// TwinCAT 3 PLC project UnitTest
// Title: TestFramework
// Company: Hoox.Software
// Author: Patrick Dressel
// ProjectVersion: 2.1.0
// ProgramVersion: 3.1.4022.6
// libraries:
//   Tc2_Standard, * (Beckhoff Automation GmbH)
//   Tc2_System, * (Beckhoff Automation GmbH)
//   Tc2_Utilities, * (Beckhoff Automation GmbH)
//   Tc3_Module, * (Beckhoff Automation GmbH)
//   Base Interfaces,newest,System
// project tree:
//   Datatypes/ EResult_t.TcDUT (not stored), EAssertion_t.TcDUT, ERetCode_t.TcDUT (not stored), EState_t.TcDUT (not stored), IdHandle_t.TcDUT (not stored), ObjectId_t.TcDUT (not stored), SStatistic_t.TcDUT (not stored), STestcase_t.TcDUT (not stored), StringHandle_t.TcDUT, StrMessage_t.TcDUT, TestCaseHandle_t.TcDUT (not stored)
//   Datatypes/Report/ EExportState_t.TcDUT (not stored), EReportType_t.TcDUT (not stored), NameHandle_t.TcDUT (not stored), PathHandle_t.TcDUT (not stored), StrFileName_t.TcDUT, StrPathName_t.TcDUT (not stored), TestReportHandle_t.TcDUT (not stored), UBaseTypes_t.TcDUT, UTime_t.TcDUT
//   GVLs/ GVL_Parameter.TcGVL (not stored), GVL_Sample.TcGVL (not stored) (excluded from build)
//   / PlcTask.TcTTO
//   Source/ FB_Assertion.TcPOU (not stored), FB_Testsuite.TcPOU (not stored), FB_TestBase.TcPOU, ITestBase_t.TcIO, ITestsuite_t.TcIO (not stored), PRG_TestLib.TcPOU
//   Source/Report/ FB_CoverageFile.TcPOU (not stored), FB_TestReportBase.TcPOU, FB_FileBase.TcPOU (not stored), FB_TextReport.TcPOU (not stored)
//   Test/ FB_Test_Base.TcPOU, FB_Test_Base_Ptr.TcPOU (not stored), FB_Test_Base_Not.TcPOU (not stored), FB_Test_Base_Delay.TcPOU

CONFIGURATION UnitTest
    RESOURCE PLC ON TwinCAT3
        TASK PlcTask(INTERVAL := T#10ms, PRIORITY := 20);
    END_RESOURCE
END_CONFIGURATION

// ---- Datatypes/EAssertion_t.TcDUT
{attribute 'qualified_only'}
{attribute 'strict'}
TYPE EAssertion_t :
(
	eStatePassed,
	eStateFailed,
	eStateFailedFatal
);
END_TYPE

// ---- Datatypes/Report/StrFileName_t.TcDUT
TYPE StrFileName_t : String(255); END_TYPE

// ---- Datatypes/Report/UBaseTypes_t.TcDUT
TYPE UBaseTypes_t :
UNION
	u8Value 	: USINT;
	s8Value 	: SINT;
	u16Value 	: UINT;
	s16Value 	: INT;
	u32Value 	: UDINT;
	s32Value 	: DINT;
	w16Value    : WORD;
	w32Value    : DWORD;
	r32Value 	: REAL;
	bValue		: BOOL;
END_UNION
END_TYPE

// ---- Datatypes/Report/UTime_t.TcDUT
TYPE UTime_t :
UNION
	dwValue  : ARRAY[0..1] OF DWORD;
	u64Value : ULINT;
END_UNION
END_TYPE

// ---- Datatypes/StringHandle_t.TcDUT
TYPE StringHandle_t : POINTER TO String(255); END_TYPE

// ---- Datatypes/StrMessage_t.TcDUT
TYPE StrMessage_t : String(255); END_TYPE

// ---- Source/ITestBase_t.TcIO
INTERFACE ITestBase_t

METHOD PUBLIC _cleanup : ERetCode_t
VAR_INPUT
END_VAR
END_METHOD

METHOD PUBLIC _execute : ERetCode_t
VAR_INPUT
END_VAR
END_METHOD

METHOD PUBLIC _prepare : ERetCode_t
VAR_INPUT
END_VAR
END_METHOD

METHOD getClassname : ObjectId_t
VAR_INPUT
END_VAR
END_METHOD

METHOD getId : ObjectId_t
VAR_INPUT
END_VAR
END_METHOD

METHOD getMessage : StrMessage_t
VAR_INPUT
END_VAR
END_METHOD

METHOD getPath : ObjectId_t
VAR_INPUT
END_VAR
END_METHOD

PROPERTY Result : STestcase_t
GET
END_GET
END_PROPERTY

END_INTERFACE

// ---- Source/FB_TestBase.TcPOU
(******************************************************************************
Baustein: FB_TestBase
Spezifikation: doc/Spezifikation.pdf, Kap. x.y.z
-------------------------------------------------------------------------------
erstellt:
von:
Geändert:
von:
-------------------------------------------------------------------------------
Beschreibung
Dieser Baustein stellt die Basis für einen Unittest dar und enthält
alle notwendigen Variablen und Methoden zur Testauswertung.

-------------------------------------------------------------------------------
Input
-

Output
	o_eResult: EResult_t;
******************************************************************************)
FUNCTION_BLOCK FB_TestBase
    IMPLEMENTS ITestBase_t
VAR_INPUT
END_VAR
VAR_OUTPUT
	o_eResult       : EResult_t;
END_VAR
VAR
	strId	  		: ObjectId_t;
	strClassName	: ObjectId_t;
	strPath			: ObjectId_t;
	strMessage 	 	: StrMessage_t;
	u32StartTime	: UDINT;
	u32EndTime		: UDINT;
	iTestSuite      : ITestsuite_t;
	bRegistered 	: BOOL;
    sResult         : STestcase_t;
    assert          : FB_Assertion;
END_VAR

(******************************************************************************
Baustein: FB_TestBase.cleanup
Spezifikation: doc/Spezifikation.pdf, Kap. x.y.z
-------------------------------------------------------------------------------
erstellt:
von:
Geändert:
von:
-------------------------------------------------------------------------------
Beschreibung
Diese Methode...

-------------------------------------------------------------------------------
Input
-

Output
-
******************************************************************************)
{attribute 'hide'} 
METHOD PUBLIC FINAL _cleanup : ERetCode_t
VAR_INPUT
END_VAR


	_cleanup := cleanup();

    IF _cleanup = ERetCode_t.eRetDone THEN
        setEndTime();
    END_IF;	
	
    CASE assert.o_eState OF 

    EAssertion_t.eStateFailed:
        o_eResult := EResult_t.eStateFailed;

    EAssertion_t.eStateFailedFatal:
        o_eResult := EResult_t.eStateFailedFatal;

    END_CASE;
END_METHOD

(******************************************************************************
Baustein: FB_TestBase.execute
Spezifikation: doc/Spezifikation.pdf, Kap. x.y.z
-------------------------------------------------------------------------------
erstellt:
von:
Geändert:
von:
-------------------------------------------------------------------------------
Beschreibung
Diese Methode...

-------------------------------------------------------------------------------
Input
-

Output
-
******************************************************************************)
{attribute 'hide'} 
METHOD PUBLIC FINAL _execute : ERetCode_t
VAR_INPUT
END_VAR

	_execute := execute();
END_METHOD

(******************************************************************************
Baustein: FB_TestBase.prepare
Spezifikation: doc/Spezifikation.pdf, Kap. x.y.z
-------------------------------------------------------------------------------
erstellt:
von:
Geändert:
von:
-------------------------------------------------------------------------------
Beschreibung
Diese Methode...

-------------------------------------------------------------------------------
Input
-

Output
-
******************************************************************************)
{attribute 'hide'} 
METHOD PUBLIC FINAL _prepare : ERetCode_t
VAR_INPUT
END_VAR

	sResult.u32Passed 		:= 0;
	sResult.u32Failed 		:= 0;
	u32StartTime 	        := 0;
	u32EndTime 		        := 0;
	o_eResult 		        := EResult_t.eStateIdle;

	_prepare := prepare();

    IF _prepare = ERetCode_t.eRetDone THEN
        setStartTime();
    END_IF;
END_METHOD

(******************************************************************************
Baustein: FB_TestBase.cleanup
Spezifikation: doc/Spezifikation.pdf, Kap. x.y.z
-------------------------------------------------------------------------------
erstellt:
von:
Geändert:
von:
-------------------------------------------------------------------------------
Beschreibung
Diese Methode...

-------------------------------------------------------------------------------
Input
-

Output
-
******************************************************************************)
METHOD PUBLIC cleanup : ERetCode_t
VAR_INPUT
END_VAR

	cleanup := ERetCode_t.eRetFailed;
END_METHOD

(******************************************************************************
Baustein: FB_TestBase.execute
Spezifikation: doc/Spezifikation.pdf, Kap. x.y.z
-------------------------------------------------------------------------------
erstellt:
von:
Geändert:
von:
-------------------------------------------------------------------------------
Beschreibung
Diese Methode...

-------------------------------------------------------------------------------
Input
-

Output
-
******************************************************************************)
METHOD PUBLIC execute : ERetCode_t
VAR_INPUT
END_VAR

	Execute := ERetCode_t.eRetFailed;
END_METHOD

(******************************************************************************
Baustein: FB_Testsuite.FB_init
Spezifikation: doc/Spezifikation.pdf, Kap. x.y.z
-------------------------------------------------------------------------------
erstellt:
von:
Geändert:
von:
-------------------------------------------------------------------------------
Beschreibung
Diese Methode

-------------------------------------------------------------------------------
Input
-

Output
-
******************************************************************************)
{attribute 'hide'} 
METHOD FB_init : BOOL
VAR_INPUT
	bInitRetains 	: BOOL; // if TRUE, the retain variables are initialized (warm start / cold start)
	bInCopyCode 	: BOOL;  // if TRUE, the instance afterwards gets moved into the copy code (online change)
	i_strId	  		: ObjectId_t;
	i_strClassName	: ObjectId_t;
	i_strPath 		: ObjectId_t;
	i_iTestSuite 	: ITestSuite_t;
	i_bExecute      : BOOL := true; 
END_VAR
	
	strId 		 := i_strId;
	strClassName := i_strClassName;
	strPath 	 := i_strPath;
	iTestSuite 	 := i_iTestSuite;

    IF i_bExecute = FALSE THEN
        o_eResult := EResult_t.eStateSkipped;
    END_IF;
	
	register();
END_METHOD

(******************************************************************************
Baustein: FB_TestBase.getId
Spezifikation: doc/Spezifikation.pdf, Kap. x.y.z
-------------------------------------------------------------------------------
erstellt:
von:
Geändert:
von:
-------------------------------------------------------------------------------
Beschreibung
Diese Methode

-------------------------------------------------------------------------------
Input
-

Output
-
******************************************************************************)
{attribute 'hide'} 
METHOD PUBLIC FINAL getClassName : ObjectId_t
VAR_INPUT
END_VAR

	getClassName := strClassName;
END_METHOD

(******************************************************************************
Baustein: FB_TestBase.getFailed
Spezifikation: doc/Spezifikation.pdf, Kap. x.y.z
-------------------------------------------------------------------------------
erstellt:
von:
Geändert:
von:
-------------------------------------------------------------------------------
Beschreibung
Diese Methode

-------------------------------------------------------------------------------
Input
-

Output
-
******************************************************************************)
{attribute 'hide'} 
METHOD PUBLIC FINAL getFailed : UDINT
VAR_INPUT
END_VAR

	getFailed := assert.o_u32Failed;
END_METHOD

(******************************************************************************
Baustein: FB_TestBase.getId
Spezifikation: doc/Spezifikation.pdf, Kap. x.y.z
-------------------------------------------------------------------------------
erstellt:
von:
Geändert:
von:
-------------------------------------------------------------------------------
Beschreibung
Diese Methode

-------------------------------------------------------------------------------
Input
-

Output
-
******************************************************************************)
{attribute 'hide'} 
METHOD PUBLIC FINAL getId : ObjectId_t
VAR_INPUT
END_VAR

	getId := strId;
END_METHOD

METHOD PUBLIC FINAL getMessage : StrMessage_t
VAR_INPUT
END_VAR

	getMessage := strMessage;
END_METHOD

(******************************************************************************
Baustein: FB_TestBase.getPassed
Spezifikation: doc/Spezifikation.pdf, Kap. x.y.z
-------------------------------------------------------------------------------
erstellt:
von:
Geändert:
von:
-------------------------------------------------------------------------------
Beschreibung
Diese Methode

-------------------------------------------------------------------------------
Input
-

Output
-
******************************************************************************)
{attribute 'hide'} 
METHOD PUBLIC FINAL getPassed : UDINT
VAR_INPUT
END_VAR

	getPassed := assert.o_u32Passed;
END_METHOD

(******************************************************************************
Baustein: FB_TestBase.getPassed
Spezifikation: doc/Spezifikation.pdf, Kap. x.y.z
-------------------------------------------------------------------------------
erstellt:
von:
Geändert:
von:
-------------------------------------------------------------------------------
Beschreibung
Diese Methode

-------------------------------------------------------------------------------
Input
-

Output
-
******************************************************************************)
{attribute 'hide'} 
METHOD PUBLIC FINAL getPath : ObjectId_t
VAR_INPUT
END_VAR

	getPath := strPath;
END_METHOD

(******************************************************************************
Baustein: FB_TestBase.getPassed
Spezifikation: doc/Spezifikation.pdf, Kap. x.y.z
-------------------------------------------------------------------------------
erstellt:
von:
Geändert:
von:
-------------------------------------------------------------------------------
Beschreibung
Diese Methode

-------------------------------------------------------------------------------
Input
-

Output
-
******************************************************************************)
{attribute 'hide'} 
METHOD PRIVATE FINAL getSystemTime : UDINT
VAR_INPUT
END_VAR
VAR
	u64Time : ULINT;
END_VAR

	u64Time := F_GetSystemTime()/10000;


	getSystemTime := to_udint(u64Time and 16#FFFFFFFF);
END_METHOD

(******************************************************************************
Baustein: FB_TestBase.getPassed
Spezifikation: doc/Spezifikation.pdf, Kap. x.y.z
-------------------------------------------------------------------------------
erstellt:
von:
Geändert:
von:
-------------------------------------------------------------------------------
Beschreibung
Diese Methode

-------------------------------------------------------------------------------
Input
-

Output
-
******************************************************************************)
{attribute 'hide'} 
METHOD PUBLIC FINAL getTime : UDINT
VAR_INPUT
END_VAR

	getTime := 0;

	IF u32EndTime > u32StartTime THEN
		getTime := u32EndTime - u32StartTime;
	END_IF;
END_METHOD

(******************************************************************************
Baustein: FB_TestBase.logError
Spezifikation: doc/Spezifikation.pdf, Kap. x.y.z
-------------------------------------------------------------------------------
erstellt:
von:
Geändert:
von:
-------------------------------------------------------------------------------
Beschreibung
Diese Methode

-------------------------------------------------------------------------------
Input
-

Output
-
******************************************************************************)
{attribute 'hide'} 
METHOD PROTECTED FINAL logError : BOOL
VAR_INPUT
	i_strMessage : StrMessage_t;
END_VAR

	ADSLOGSTR(msgCtrlMask 	:= ADSLOG_MSGTYPE_ERROR , 
			  msgFmtStr 	:= i_strMessage, 
			  strArg 		:= '');
END_METHOD

(******************************************************************************
Baustein: FB_TestBase.logInfo
Spezifikation: doc/Spezifikation.pdf, Kap. x.y.z
-------------------------------------------------------------------------------
erstellt:
von:
Geändert:
von:
-------------------------------------------------------------------------------
Beschreibung
Diese Methode

-------------------------------------------------------------------------------
Input
-

Output
-
******************************************************************************)
{attribute 'hide'} 
METHOD INTERNAL FINAL logInfo : BOOL
VAR_INPUT
	i_strMessage : StrMessage_t;
END_VAR

	ADSLOGSTR(msgCtrlMask 	:= ADSLOG_MSGTYPE_HINT , 
			  msgFmtStr 	:= i_strMessage, 
			  strArg 		:= '');
END_METHOD

(******************************************************************************
Baustein: FB_TestBase.prepare
Spezifikation: doc/Spezifikation.pdf, Kap. x.y.z
-------------------------------------------------------------------------------
erstellt:
von:
Geändert:
von:
-------------------------------------------------------------------------------
Beschreibung
Diese Methode...

-------------------------------------------------------------------------------
Input
-

Output
-
******************************************************************************)
METHOD PUBLIC prepare : ERetCode_t
VAR_INPUT
END_VAR

	prepare := ERetCode_t.eRetFailed;
END_METHOD

(******************************************************************************
Baustein: FB_TestBase.register
Spezifikation: doc/Spezifikation.pdf, Kap. x.y.z
-------------------------------------------------------------------------------
erstellt:
von:
Geändert:
von:
-------------------------------------------------------------------------------
Beschreibung
Diese Methode

-------------------------------------------------------------------------------
Input
-

Output
-
******************************************************************************)
{attribute 'hide'} 
METHOD INTERNAL FINAL register : BOOL
VAR_INPUT
END_VAR

	IF iTestSuite <> 0 	AND 
       bRegistered = FALSE  THEN
		
	   bRegistered := iTestSuite.addTestcase(THIS^);
	
	END_IF
END_METHOD

{warning 'Eigenschaftenimplementierung hinzufügen'}
PROPERTY Result : STestcase_t
GET

    sResult.u32Time := getTime();
    sResult.eState  := o_eResult; 
    Result          := sResult;
END_GET
END_PROPERTY

(******************************************************************************
Baustein: FB_TestBase.getPassed
Spezifikation: doc/Spezifikation.pdf, Kap. x.y.z
-------------------------------------------------------------------------------
erstellt:
von:
Geändert:
von:
-------------------------------------------------------------------------------
Beschreibung
Diese Methode

-------------------------------------------------------------------------------
Input
-

Output
-
******************************************************************************)
{attribute 'hide'} 
METHOD INTERNAL FINAL setEndTime : BOOL
VAR_INPUT
END_VAR

	IF u32EndTime = 0 THEN
		u32EndTime := getSystemTime();
	END_IF;
	setEndTime := true;
END_METHOD

METHOD PROTECTED FINAL setMessage
VAR_INPUT
	strValue : StrMessage_t;
END_VAR

	IF o_eResult < EResult_t.eStateFailed THEN
		strMessage := strValue;
	END_IF;
END_METHOD

(******************************************************************************
Baustein: FB_TestBase.getPassed
Spezifikation: doc/Spezifikation.pdf, Kap. x.y.z
-------------------------------------------------------------------------------
erstellt:
von:
Geändert:
von:
-------------------------------------------------------------------------------
Beschreibung
Diese Methode

-------------------------------------------------------------------------------
Input
-

Output
-
******************************************************************************)
{attribute 'hide'} 
METHOD INTERNAL FINAL setStartTime : BOOL
VAR_INPUT
END_VAR

	IF u32StartTime = 0 THEN
		u32StartTime   	:= getSystemTime();
	END_IF;
	setStartTime := true;
END_METHOD

(******************************************************************************
Baustein: FB_TestBase.strncmp
Spezifikation: doc/Spezifikation.pdf, Kap. x.y.z
-------------------------------------------------------------------------------
erstellt:
von:
Geändert:
von:
-------------------------------------------------------------------------------
Beschreibung
Diese Methode

-------------------------------------------------------------------------------
Input
	strInput 	: StringHandle_t;
	strCompare 	: StringHandle_t;
	s16Size		: INT;

Output
-
******************************************************************************)
{attribute 'hide'} 
METHOD PRIVATE FINAL strncmp : BOOL
VAR_INPUT
	strInput 	: StringHandle_t;
	strCompare 	: StringHandle_t;
	s16Size		: INT;
END_VAR
VAR
	s16Size1 : INT;
	s16Size2 : INT;
	s16Diff  : INT;
END_VAR

   s16Size1:= LEN(strInput^); 
	s16Size2:= LEN(strCompare^); 
	
	strncmp := FALSE;
	
	s16Diff := s16Size1 - s16Size2;
   
	// vergleich nur wenn beide Strings
	// gleich groß sind.
	IF s16Diff  = 0 THEN

		strncmp := TRUE;
	
		WHILE(s16Size > 0) DO

			IF strInput^ <> strCompare^ THEN
				strncmp := FALSE;
			END_IF;  
 
			strInput   := strInput + 1;
			strCompare := strCompare + 1;
			s16Size    := s16Size - 1;

		END_WHILE


	
	END_IF;
END_METHOD

(******************************************************************************
Baustein: FB_TestBase.validate
Spezifikation: doc/Spezifikation.pdf, Kap. x.y.z
-------------------------------------------------------------------------------
erstellt:
von:
Geändert:
von:
-------------------------------------------------------------------------------
Beschreibung
Diese Methode

-------------------------------------------------------------------------------
Input
	var1 : ANY;
	var2 : ANY;

Output
-
******************************************************************************)
{attribute 'hide'} 
METHOD PRIVATE FINAL validate : BOOL
VAR_INPUT
	var1 : ANY;
	var2 : ANY;
END_VAR

	validate := FALSE;
	
	IF (var1.pValue = 0 OR var2.pValue = 0) THEN
		logError(concat('Assert validation fails with NULL-Pointer: ', strId));
		RETURN;
	END_IF

	IF (var1.TypeClass <> var2.TypeClass) THEN
		logError(concat('Assert validation fails with TypeClass Error: ', strId));
		RETURN;
	END_IF;	
	
	IF (var1.diSize <> var2.diSize) THEN
		logError(concat('Assert validation fails with different size: ', strId));
		RETURN;
	END_IF;	
	
	validate := true;
END_METHOD

END_FUNCTION_BLOCK

// ---- Source/PRG_TestLib.TcPOU
(******************************************************************************
Baustein: PRG_TestLibrary
Spezifikation: doc/Spezifikation.pdf, Kap. x.y.z
-------------------------------------------------------------------------------
erstellt:
von:
Geändert:
von:
-------------------------------------------------------------------------------
Beschreibung
Dieser Baustein etnhält alle Testsuites und führt diese aus.

-------------------------------------------------------------------------------
Input
	i_bStart : mit positiver Flanke werden die registrierten Testsuites ausgeführt

Output
	o_eState  		: EState_t;
	o_eResult 		: EResult_t;
	o_sStatistic	: SStatistic_t;
******************************************************************************)
{attribute 'global_init_slot' := '41000'}
PROGRAM PRG_TestLib
VAR_INPUT
	i_bStart : BOOL;
END_VAR
VAR_OUTPUT
	o_eState  		: EState_t;
	o_eResult 		: EResult_t;
	o_sStatistic	: SStatistic_t;
END_VAR
VAR
	bHwStart AT %I* : BOOL;
	bHwBusy  AT %Q* : BOOL;
	bHwReady AT %Q* : BOOL;
	
	a_iTestSuite 	: ARRAY [0..255] OF ITestSuite_t;
	u16TestSuites 	: UINT;
	u16Index	  	: UINT;
	iActTestSuite 	: ITestSuite_t;
	pTestReport		: POINTER TO FB_TestReportBase;
	eRetCode 		: ERetCode_t;

	fbSystemTime 	: FB_LocalSystemTime;
	
	fbUnittest 		: FB_CoverageFile;
	u16ReportState  : UINT;
	u16TestSuitIdx	: UINT;
	iTestCase  		: ITestBase_t;
	sTempResult     : SStatistic_t;
END_VAR
VAR CONSTANT 
END_VAR


	fbSystemTime(bEnable := TRUE, dwCycle := 5);
			
	fbUnittest();

	CASE o_eState OF 
	
	EState_t.eStateInit:	
		
		IF i_bStart = FALSE THEN 
		   logInfo('Testlib V2.1.0 Ready');
			o_eState := EState_t.eStateIdle; 
		END_IF

	EState_t.eStateIdle:
	
		IF i_bStart = TRUE OR bHwStart = TRUE THEN
			logInfo('+++++++++++++ Testbeginn ++++++++++++++');
			o_eState := EState_t.eStatePrepare;
			bHwReady := FALSE;
		END_IF
	
	EState_t.eStatePrepare:
	
		bHwBusy := TRUE;
		
		o_eResult 	  				:= EResult_t.eStatePassed;
		o_sStatistic.u32Executed 	:= 0;
		o_sStatistic.u32TestCases	:= 0;
		o_sStatistic.u32Asserts  	:= 0;
		o_sStatistic.u32Passed   	:= 0;
		o_sStatistic.u32Failed	 	:= 0;	

		iActTestSuite := getFirstTestSuite();
		
		IF iActTestSuite      <> 0   THEN
			o_eState := EState_t.eStateExecute;
		ELSE
			o_eState := EState_t.eStateError;	
		END_IF
	
	EState_t.eStateExecute:
	
		iActTestSuite.execute(i_bStart := TRUE);
	
		IF iActTestSuite.getState() = EState_t.eStateReady THEN
			
			IF iActTestSuite.getResult() = EResult_t.eStateFailed THEN
				o_eResult := EResult_t.eStateFailed;
			END_IF
			
			iActTestSuite.execute(i_bStart := FALSE);
			sTempResult := iActTestSuite.Result;

			o_eState := EState_t.eStateCleanUp;

			o_sStatistic.u32Executed 	:= o_sStatistic.u32Executed  + sTempResult.u32Executed;
			o_sStatistic.u32TestCases	:= o_sStatistic.u32TestCases + sTempResult.u32TestCases; 
			o_sStatistic.u32Asserts  	:= o_sStatistic.u32Asserts   + sTempResult.u32Asserts;
			o_sStatistic.u32Passed   	:= o_sStatistic.u32Passed    + sTempResult.u32Passed;
			o_sStatistic.u32Failed	 	:= o_sStatistic.u32Failed    + sTempResult.u32Failed;
		END_IF
	
	EState_t.eStateCleanUp:
	
		IF iActTestSuite.getResult() = EResult_t.eStateFailedFatal THEN
			o_eResult := EResult_t.eStateFailedFatal;
			o_eState  := EState_t.eStateExport;
			logInfo('+++++++++++++ Fatal Error : Test Ende ++++++++++++++');
		ELSE
			
			iActTestSuite := getNextTestSuite();
						
			IF iActTestSuite <> 0 THEN
				o_eState := EState_t.eStateExecute;
			ELSE
				o_eState := EState_t.eStateExport;
				logInfo('+++++++++++++ Test Ende ++++++++++++++');
			END_IF		
			
		END_IF

	EState_t.eStateExport:

		IF createReport(EReporttype_t.eExternalReport) = ERetCode_t.eRetDone THEN
			o_eState := EState_t.eStateBuildUnitTestFile;
		END_IF;
		
	EState_t.eStateBuildUnitTestFile:

		IF createReport(EReporttype_t.eUnitTestReport) = ERetCode_t.eRetDone THEN
			o_eState := EState_t.eStateReady;
		END_IF;
		
	EState_t.eStateReady:

		bHwReady := TRUE;
		bHwBusy  := FALSE;
		IF i_bStart  = FALSE AND 
			bHwStart = FALSE THEN
			o_eState := EState_t.eStateIdle;
		END_IF		
		
	EState_t.eStateError,
	EState_t.eStateLicenseError:
	
		bHwBusy  := FALSE;
		o_eState := EState_t.eStateError;

	END_CASE

(******************************************************************************
Baustein: PRG_UnitTestLib.addTestReport
Spezifikation: doc/Spezifikation.pdf, Kap. x.y.z
-------------------------------------------------------------------------------
erstellt:
von:
Geändert:
von:
-------------------------------------------------------------------------------
Beschreibung
Diese Methode

-------------------------------------------------------------------------------
Input
i_pTestReport

Output
-
******************************************************************************)
{attribute 'hide'} 
METHOD PUBLIC addTestReport : BOOL
VAR_INPUT
	i_pTestReport : TestReportHandle_t;
END_VAR

	pTestReport := i_pTestReport;
END_METHOD

(******************************************************************************
Baustein: PRG_UnitTestLib.addTestSuite
Spezifikation: doc/Spezifikation.pdf, Kap. x.y.z
-------------------------------------------------------------------------------
erstellt:
von:
Geändert:
von:
-------------------------------------------------------------------------------
Beschreibung
Diese Methode

-------------------------------------------------------------------------------
Input
i_pTestSuite

Output
-
******************************************************************************)
{attribute 'hide'} 
METHOD PUBLIC addTestSuite : BOOL
VAR_INPUT
	i_iTestSuite : ITestSuite_t;
END_VAR
VAR
    sStatistic : SStatistic_t;
END_VAR

	addTestSuite := FALSE;

	IF 	i_iTestSuite  <> 0   AND 
		u16TestSuites <  255 THEN
		
		a_iTestSuite[u16TestSuites] := i_iTestSuite;
		sStatistic      := i_iTestSuite.Result;
		u16TestSuites   := u16TestSuites +1;
	
		o_sStatistic.u32TestSuites := o_sStatistic.u32TestSuites + 1;
		o_sStatistic.u32TestCases  := o_sStatistic.u32TestCases + sStatistic.u32TestCases;
		
		addTestSuite := TRUE;
	END_IF
END_METHOD

{attribute 'hide'} 
METHOD PRIVATE createReport : ERetCode_t
VAR_INPUT
	i_eReporttype : EReportType_t;
END_VAR
VAR
	eRetcode    : ERetCode_t;
	u32Temp     : UDINT;
    sTestResult : STestcase_t;
    sStatistic  : SStatistic_t;
END_VAR

	createReport := ERetCode_t.eRetBusy;

	CASE u16ReportState OF

	0: 
		IF i_eReporttype = EReportType_t.eUnitTestReport THEN
			u16ReportState := 20;
		END_IF;

		IF i_eReporttype = EReportType_t.eExternalReport THEN
			u16ReportState := 100;
		END_IF;

// +++++++++++++++++++++++++++++++++++++++++++++++++++++++++++
//
// Export Unittest Ergebnisse
// 
// +++++++++++++++++++++++++++++++++++++++++++++++++++++++++++
	20:		

		eRetcode := fbUnitTest.open('C:\TwinCAT\3.1\Boot\CurrentConfig\', 'Unittest.xml');

		IF eRetcode = ERetCode_t.eRetDone THEN

			u16ReportState := 21;

		ELSIF eRetcode = ERetCode_t.eRetFailed THEN

			logError('createReport Unittest.xml : Datei nicht geöffnet');
			u16ReportState := 22;

		END_IF;	

	21:

		u16TestSuitIdx := 0;

		fbUnitTest.addString('<?xml version="1.0" ?>');
		fbUnitTest.addCrlf();

		iActTestSuite := getFirstTestSuite();

		WHILE (iActTestSuite <> 0) DO

            sStatistic := iActTestSuite.Result;
			u16TestSuitIdx := u16TestSuitIdx+1;

			fbUnitTest.addString('<testsuite');
			fbUnitTest.addString(' name="');
			fbUnitTest.addString(iActTestSuite.getId());
			fbUnitTest.addString('" tests="');			
			fbUnitTest.addValue(sStatistic.u32TestCases);
			fbUnitTest.addString('" disabled="');
            u32Temp := sStatistic.u32TestCases-sStatistic.u32Executed;
			fbUnitTest.addValue(u32Temp);
			fbUnitTest.addString('" errors="');
			fbUnitTest.addValue(u32Temp);
			fbUnitTest.addString('" failures="');
			fbUnitTest.addValue(sStatistic.u32Failed);
			fbUnitTest.addString('" hostname="');
			fbUnitTest.addString('" id="');
			fbUnitTest.addvalue(u16TestSuitIdx);
			fbUnitTest.addString('" package="');
			fbUnitTest.addString(iActTestSuite.getPath());
			fbUnitTest.addString('">');
			fbUnitTest.addCrlf();

			iTestCase := iActTestSuite.getFirstTestCase();

			WHILE (iTestCase <> 0) DO
        
                sTestResult := iTestCase.Result;

				fbUnitTest.addString('<testcase');
				fbUnitTest.addString(' name="');
				fbUnitTest.addString(iTestCase.getId());
				fbUnitTest.addString('" assertions="');
                u32Temp := sTestResult.u32Failed + sTestResult.u32Passed;
				fbUnitTest.addValue(u32Temp);
				fbUnitTest.addString('" classname="');
				fbUnitTest.addString(iTestCase.getPath());
                fbUnitTest.addString('.');
				fbUnitTest.addString(iTestCase.getClassName());
				fbUnitTest.addString('" time="');				
				fbUnitTest.addTimeMs(sTestResult.u32Time);
				fbUnitTest.addString('">');
				fbUnitTest.addCrlf();

				CASE sTestResult.eState OF

				EResult_t.eStatePassed :

					fbUnitTest.addString('<passed/>');

				EResult_t.eStateFailed, 
				EResult_t.eStateFailedFatal :
			
					fbUnitTest.addString('<failure');
					fbUnitTest.addString(' message="');
					fbUnitTest.addString(iTestCase.getMessage());
					fbUnitTest.addString('"/>');
					
				EResult_t.eStateSkipped:

					fbUnitTest.addString('<skipped/>');

				END_CASE;
				
				fbUnitTest.addCrlf();	

				fbUnitTest.addString('</testcase>');
				fbUnitTest.addCrlf();		

				iTestCase := iActTestSuite.getNextTestCase();
		
			END_WHILE

			fbUnitTest.addString('</testsuite>');
			fbUnitTest.addCrlf();	

			iActTestSuite := getNextTestSuite();

		END_WHILE

		fbUnitTest.addString('</testsuites>');
		fbUnitTest.addCrlf();

		u16ReportState := 22;

	22:
		IF fbUnitTest.o_bOpen  = TRUE AND 
		   fbUnitTest.o_bEmpty = TRUE THEN
			fbUnitTest.close();
		END_IF;

		IF fbUnitTest.o_bOpen  = FALSE THEN
			createReport 	:= ERetCode_t.eRetDone;
		END_IF;

// +++++++++++++++++++++++++++++++++++++++++++++++++++++++++++
//
//
// 
// +++++++++++++++++++++++++++++++++++++++++++++++++++++++++++
	100:

		IF pTestReport <> 0 THEN
			
			createReport := pTestReport^.create();		
			
		ELSE

			createReport := ERetCode_t.eRetDone;

		END_IF;

	ELSE
		createReport := ERetCode_t.eRetFailed;
	END_CASE;

	IF createReport = ERetCode_t.eRetDone THEN
		u16ReportState := 0;
	END_IF;
















(**)
END_METHOD

(******************************************************************************
Baustein: PRG_UnitTestLib.getFirstTestSuite
Spezifikation: doc/Spezifikation.pdf, Kap. x.y.z
-------------------------------------------------------------------------------
erstellt:
von:
Geändert:
von:
-------------------------------------------------------------------------------
Beschreibung
Diese Methode

-------------------------------------------------------------------------------
Input
-

Output
-
******************************************************************************)
{attribute 'hide'} 
METHOD PRIVATE getFirstTestSuite : ITestSuite_t
VAR_INPUT
END_VAR

	u16Index := 0;
	getFirstTestSuite := a_iTestSuite[0];
END_METHOD

(******************************************************************************
Baustein: PRG_UnitTestLib.getNextTestSuite
Spezifikation: doc/Spezifikation.pdf, Kap. x.y.z
-------------------------------------------------------------------------------
erstellt:
von:
Geändert:
von:
-------------------------------------------------------------------------------
Beschreibung
Diese Methode

-------------------------------------------------------------------------------
Input
-

Output
-
******************************************************************************)
{attribute 'hide'} 
METHOD PRIVATE getNextTestSuite : ITestSuite_t
VAR_INPUT
END_VAR

	getNextTestSuite := 0;
	u16Index 		 := u16Index + 1;

	IF u16Index < u16TestSuites THEN
		getNextTestSuite := a_iTestSuite[u16Index];
	END_IF;
END_METHOD

(******************************************************************************
Baustein: PRG_UnitTestLib.getTime
Spezifikation: doc/Spezifikation.pdf, Kap. x.y.z
-------------------------------------------------------------------------------
erstellt:
von:
Geändert:
von:
-------------------------------------------------------------------------------
Beschreibung
Diese Methode

-------------------------------------------------------------------------------
Input
-

Output
-
******************************************************************************)
{attribute 'hide'} 
METHOD getTime : TimeStruct
VAR_INPUT
END_VAR
VAR
END_VAR

	getTime := fbSystemTime.systemTime;
END_METHOD

(******************************************************************************
Baustein: PRG_UnitTestLib.logError
Spezifikation: doc/Spezifikation.pdf, Kap. x.y.z
-------------------------------------------------------------------------------
erstellt:
von:
Geändert:
von:
-------------------------------------------------------------------------------
Beschreibung
Diese Methode

-------------------------------------------------------------------------------
Input
i_strMessage

Output
-
******************************************************************************)
{attribute 'hide'} 
METHOD PROTECTED logError : BOOL
VAR_INPUT
	i_strMessage : StrMessage_t;
END_VAR

	ADSLOGSTR(msgCtrlMask 	:= ADSLOG_MSGTYPE_ERROR , 
			  msgFmtStr 	:= i_strMessage, 
			  strArg 		:= '');
END_METHOD

(******************************************************************************
Baustein: PRG_UnitTestLib.logInfo
Spezifikation: doc/Spezifikation.pdf, Kap. x.y.z
-------------------------------------------------------------------------------
erstellt:
von:
Geändert:
von:
-------------------------------------------------------------------------------
Beschreibung
Diese Methode

-------------------------------------------------------------------------------
Input
i_strMessage

Output
-
******************************************************************************)
{attribute 'hide'} 
METHOD PUBLIC logInfo : BOOL
VAR_INPUT
	i_strMessage : StrMessage_t;
END_VAR

	ADSLOGSTR(msgCtrlMask 	:= ADSLOG_MSGTYPE_HINT , 
			  msgFmtStr 	:= i_strMessage, 
			  strArg 		:= '');
END_METHOD

END_PROGRAM

// ---- Source/Report/FB_TestReportBase.TcPOU
(******************************************************************************
Baustein: FB_TestReportBase
Spezifikation: doc/Spezifikation.pdf, Kap. x.y.z
-------------------------------------------------------------------------------
erstellt:
von:
Geändert:
von:
-------------------------------------------------------------------------------
Beschreibung
Dieser Baustein enthält alle zugeordneten Testfälle. Ein Testfall
ist ein abgeleiteter Baustein (FB) von FB_UnitTestBase.

-------------------------------------------------------------------------------
Input
-

Output
-
******************************************************************************)
FUNCTION_BLOCK FB_TestReportBase
VAR_INPUT
END_VAR
VAR_OUTPUT
END_VAR
VAR
	strBuffer   : STRING(255);
	fbOpen      : FB_FileOpen;
	fbClose     : FB_FileClose;
	fbWrite	    : FB_FileWrite;
	strFileName : StrFileName_t;
	strFilePath : StrPathName_t;
	
	eState 		: EExportState_t;
	u32Line     : UDINT;
	
	sStatistic  : SStatistic_t;

	trgOpen 	: F_TRIG;
	trgWrite 	: F_TRIG;
	trgClose 	: F_TRIG;
END_VAR

(******************************************************************************
Baustein: FB_TestReportBase.addCrlf
Spezifikation: doc/Spezifikation.pdf, Kap. x.y.z
-------------------------------------------------------------------------------
erstellt:
von:
Geändert:
von:
-------------------------------------------------------------------------------
Beschreibung


-------------------------------------------------------------------------------
Input
-

Output
-
******************************************************************************)
METHOD PROTECTED addCrlf : BOOL
VAR_INPUT
END_VAR
VAR
END_VAR
   
	strBuffer := CONCAT(strBuffer, '$R$N');
END_METHOD

(******************************************************************************
Baustein: FB_TestReportBase.addDate
Spezifikation: doc/Spezifikation.pdf, Kap. x.y.z
-------------------------------------------------------------------------------
erstellt:
von:
Geändert:
von:
-------------------------------------------------------------------------------
Beschreibung

-------------------------------------------------------------------------------
Input
	i_sDate : TIMESTRUCT;

Output
-
******************************************************************************)
METHOD PROTECTED addDate : ERetCode_t
VAR_INPUT
	i_sDate : TIMESTRUCT;
END_VAR

   	addDate := ERetcode_t.eRetDone;

   	addValue(i_sDate.wDay);
   	addString('.');
   	addValue(i_sDate.wMonth);
   	addString('.');
    addValue(i_sDate.wYear);
    addString(' ');
END_METHOD

(******************************************************************************
Baustein: FB_TestReportBase.addString
Spezifikation: doc/Spezifikation.pdf, Kap. x.y.z
-------------------------------------------------------------------------------
erstellt:
von:
Geändert:
von:
-------------------------------------------------------------------------------
Beschreibung

-------------------------------------------------------------------------------
Input
	i_strData : STRING(255);

Output
-
******************************************************************************)
METHOD PROTECTED addString : ERetCode_t
VAR_INPUT
	i_strData : STRING(255);
END_VAR

	strBuffer :=  concat(strBuffer, i_strData);

	addString := ERetcode_t.eRetDone;
END_METHOD

(******************************************************************************
Baustein: FB_TestReportBase.addTime
Spezifikation: doc/Spezifikation.pdf, Kap. x.y.z
-------------------------------------------------------------------------------
erstellt:
von:
Geändert:
von:
-------------------------------------------------------------------------------
Beschreibung

-------------------------------------------------------------------------------
Input
	i_sTime : TIMESTRUCT;

Output
-
******************************************************************************)
METHOD PROTECTED addTime : ERetCode_t
VAR_INPUT
	i_sTime : TIMESTRUCT;
END_VAR

	addTime := ERetcode_t.eRetDone;
	
   	addValue(i_sTime.wHour);
   	addString('.');
   	addValue(i_sTime.wMinute);
  	addString('.');
   	addValue(i_sTime.wSecond);
   	addString(' ');
END_METHOD

(******************************************************************************
Baustein: FB_TestReportBase.addValue
Spezifikation: doc/Spezifikation.pdf, Kap. x.y.z
-------------------------------------------------------------------------------
erstellt:
von:
Geändert:
von:
-------------------------------------------------------------------------------
Beschreibung

-------------------------------------------------------------------------------
Input
	i_anyValue : ANY;

Output
-
******************************************************************************)
METHOD PROTECTED addValue : ERetCode_t
VAR_INPUT
	i_anyValue : ANY;
END_VAR
VAR
	uValue : UBaseTypes_t;
END_VAR

	addValue  := ERetcode_t.eRetDone;
	
	IF i_anyValue.pValue = 0 THEN
		addValue  := ERetcode_t.eRetFailed;
		RETURN;
	END_IF

	MEMCPY(ADR(uValue),i_anyValue.pValue, TO_UDINT(i_anyValue.diSize)); 

	CASE i_anyValue.TypeClass OF

	IBaseLibrary.TYPE_SINT:

		addString(SINT_TO_STRING(uValue.s8Value));

	//IBaseLibrary.TYPE_BYTE:
	IBaseLibrary.TYPE_USINT:

		addString(USINT_TO_STRING(uValue.u8Value));

	IBaseLibrary.TYPE_INT:

		addString(INT_TO_STRING(uValue.s16Value));

	IBaseLibrary.TYPE_DINT:

		addString(DINT_TO_STRING(uValue.s32Value));

	IBaseLibrary.TYPE_UINT:

		addString(UINT_TO_STRING(uValue.u16Value));

	IBaseLibrary.TYPE_UDINT:

		addString(UDINT_TO_STRING(uValue.u32Value));

	IBaseLibrary.TYPE_WORD:

		addString(WORD_TO_STRING(uValue.w16Value));

	IBaseLibrary.TYPE_DWORD:

		addString(DWORD_TO_STRING(uValue.w32Value));

	ELSE
		ADSLOGSTR(msgCtrlMask 	:= ADSLOG_MSGTYPE_ERROR , 
				  msgFmtStr 	:= 'TestReportBase.AddValue: Unbekannter Datentyp!', 
				  strArg 		:= '');
	END_CASE;
END_METHOD

(******************************************************************************
Baustein: FB_TestReportBase.BuildFile
Spezifikation: doc/Spezifikation.pdf, Kap. x.y.z
-------------------------------------------------------------------------------
erstellt:
von:
Geändert:
von:
-------------------------------------------------------------------------------
Beschreibung
Diese Methode muss vom ableitenden Baustein überschrieben werden und
wird von der Basisklasse aus aufgerufen wenn der Report erstellt werden
soll.

-------------------------------------------------------------------------------
Input
-

Output
-
******************************************************************************)
METHOD PROTECTED BuildFile : ERetCode_t
VAR_INPUT
	i_u32Line : UDINT;
END_VAR
END_METHOD

(******************************************************************************
Baustein: FB_TestReportBase.clearBuffer
Spezifikation: doc/Spezifikation.pdf, Kap. x.y.z
-------------------------------------------------------------------------------
erstellt:
von:
Geändert:
von:
-------------------------------------------------------------------------------
Beschreibung

-------------------------------------------------------------------------------
Input
-

Output
-
******************************************************************************)
METHOD PROTECTED clearBuffer : ERetCode_t
VAR_INPUT
END_VAR

	clearBuffer := ERetCode_t.eRetDone;
	
	strBuffer := '';
END_METHOD

(******************************************************************************
Baustein: FB_TestReportBase.Close
Spezifikation: doc/Spezifikation.pdf, Kap. x.y.z
-------------------------------------------------------------------------------
erstellt:
von:
Geändert:
von:
-------------------------------------------------------------------------------
Beschreibung


-------------------------------------------------------------------------------
Input
-

Output
-
******************************************************************************)
METHOD PROTECTED Close : ERetCode_t
VAR_INPUT
END_VAR

	Close := ERetCode_t.eRetFailed;
	
	fbClose.hFile 		:= fbOpen.hFile;
	fbClose.bExecute 	:= TRUE; 

	IF trgClose.Q = TRUE THEN
		Close := ERetCode_t.eRetDone;
		fbClose.bExecute  := FALSE;		
	ELSE	
		Close := ERetCode_t.eRetBusy;
	END_IF;	
	
	IF fbClose.bError = TRUE THEN
		Close := eRetCode_t.eRetFailed;
	END_IF;
END_METHOD

(******************************************************************************
Baustein: FB_TestReportBase.create
Spezifikation: doc/Spezifikation.pdf, Kap. x.y.z
-------------------------------------------------------------------------------
erstellt:
von:
Geändert:
von:
-------------------------------------------------------------------------------
Beschreibung


-------------------------------------------------------------------------------
Input
-

Output
-
******************************************************************************)
METHOD PUBLIC create : ERetCode_t;
VAR_INPUT
END_VAR
VAR
	eRetCode : ERetCode_t;
END_VAR

	create := ERetCode_t.eRetBusy;

	fbOpen();
	fbWrite();
	fbClose();

	trgOpen(CLK := fbOpen.bBusy);
	trgWrite(CLK := fbWrite.bBusy);
	trgClose(CLK := fbClose.bBusy);
	
	CASE eState OF
	
	EExportState_t.eExportIdle:
	
		eState := EExportState_t.eExportOpen;
	
	EExportState_t.eExportOpen:
	
		eRetCode 	:= Open();
		u32Line  	:= 0;
		sStatistic 	:= PRG_UnitTestLib.o_sStatistic;

		IF eRetCode = ERetCode_t.eRetDone THEN
			eState := EExportState_t.eExportGetLine;
		ELSIF eRetCode = ERetCode_t.eRetFailed THEN
			eState := EExportState_t.eExportError;
		END_IF;

	EExportState_t.eExportGetLine:

		eRetCode := BuildFile(u32Line);

		IF eRetCode = ERetCode_t.eRetDone THEN
			eState := EExportState_t.eExportClose;
		ELSIF eRetCode = ERetCode_t.eRetFailed THEN
			eState := EExportState_t.eExportError;
		ELSE
			addCrlf();
			eState := EExportState_t.eExportWrite;
		END_IF;

	EExportState_t.eExportWrite:
	
		IF writeBuffer() =  ERetCode_t.eRetDone THEN
			clearBuffer();	
			u32Line := u32Line + 1;
			eState  := EExportState_t.eExportGetLine;
		END_IF;		
	
	EExportState_t.eExportClose:
	
		eRetCode := Close();
		
		IF eRetCode = ERetCode_t.eRetDone THEN
			eState     := EExportState_t.eExportIdle;
			create	   := ERetCode_t.eRetDone;
			reset();
		ELSIF eRetCode = ERetCode_t.eRetFailed THEN
			eState := EExportState_t.eExportError;
		end_if;
	
	EExportState_t.eExportError:
	
		create := ERetCode_t.eRetFailed;
	
	end_case;
END_METHOD

(******************************************************************************
Baustein: FB_TestReportBase.FB_Init
Spezifikation: doc/Spezifikation.pdf, Kap. x.y.z
-------------------------------------------------------------------------------
erstellt:
von:
Geändert:
von:
-------------------------------------------------------------------------------
Beschreibung


-------------------------------------------------------------------------------
Input
-

Output
-
******************************************************************************)
METHOD FB_init : BOOL
VAR_INPUT
	bInitRetains : BOOL; // if TRUE, the retain variables are initialized (warm start / cold start)
	bInCopyCode : BOOL;  // if TRUE, the instance afterwards gets moved into the copy code (online change)
END_VAR

	PRG_UnitTestLib.addTestReport(this);
END_METHOD

(******************************************************************************
Baustein: FB_TestReportBase.getFileName
Spezifikation: doc/Spezifikation.pdf, Kap. x.y.z
-------------------------------------------------------------------------------
erstellt:
von:
Geändert:
von:
-------------------------------------------------------------------------------
Beschreibung
Diese Methode muss vom ableitenden Baustein überschrieben werden und
wird von der Basisklasse aus aufgerufen wenn der Report erstellt werden
soll.

-------------------------------------------------------------------------------
Input
	i_pFileName : NameHandle_t;
	i_pPath		: PathHandle_t;

Output
-
******************************************************************************)
METHOD PROTECTED getFileName : ERetCode_t
VAR_INPUT
	i_pFileName : NameHandle_t;
	i_pPath		: PathHandle_t;
END_VAR
END_METHOD

(******************************************************************************
Baustein: FB_TestReportBase.getTime
Spezifikation: doc/Spezifikation.pdf, Kap. x.y.z
-------------------------------------------------------------------------------
erstellt:
von:
Geändert:
von:
-------------------------------------------------------------------------------
Beschreibung


-------------------------------------------------------------------------------
Input
-

Output
-
******************************************************************************)
METHOD PROTECTED getTime : TimeStruct
VAR_INPUT
END_VAR
VAR
END_VAR

	getTime := PRG_UnitTestLib.getTime();
END_METHOD

(******************************************************************************
Baustein: FB_TestReportBase.Open
Spezifikation: doc/Spezifikation.pdf, Kap. x.y.z
-------------------------------------------------------------------------------
erstellt:
von:
Geändert:
von:
-------------------------------------------------------------------------------
Beschreibung


-------------------------------------------------------------------------------
Input
-

Output
-
******************************************************************************)
METHOD PROTECTED open : ERetCode_t
VAR_INPUT
END_VAR

	open := ERetCode_t.eRetFailed;

	getFileName(ADR(strFileName), ADR(strFilePath));
	
	fbOpen.sPathName := CONCAT(strFilePath, strFileName);
	fbOpen.nMode 	 := FOPEN_MODEWRITE OR FOPEN_MODEBINARY;	
	fbOpen.bExecute  := TRUE;
			
	IF trgOpen.Q = TRUE THEN
		open := ERetCode_t.eRetDone;
		fbOpen.bExecute  := FALSE;		
	ELSE	
		open := ERetCode_t.eRetBusy;
	END_IF;	
	
	IF fbOpen.bError = TRUE THEN
		open := eRetCode_t.eRetFailed;
	END_IF;
END_METHOD

(******************************************************************************
Baustein: FB_TestReportBase.reset
Spezifikation: doc/Spezifikation.pdf, Kap. x.y.z
-------------------------------------------------------------------------------
erstellt:
von:
Geändert:
von:
-------------------------------------------------------------------------------
Beschreibung


-------------------------------------------------------------------------------
Input
-

Output
-
******************************************************************************)
METHOD PUBLIC reset : BOOL
VAR_INPUT
END_VAR

	IF fbOpen.hFile <> 0 THEN
		close();
	END_IF
	
	clearBuffer();

	fbOpen(sPathName := '', bExecute := FALSE);
	
	fbWrite(bExecute := FALSE);
	
	fbClose(bExecute := FALSE);
	
	eState := EExportState_t.eExportIdle;
END_METHOD

(******************************************************************************
Baustein: FB_TestReportBase.writeBuffer
Spezifikation: doc/Spezifikation.pdf, Kap. x.y.z
-------------------------------------------------------------------------------
erstellt:
von:
Geändert:
von:
-------------------------------------------------------------------------------
Beschreibung


-------------------------------------------------------------------------------
Input
-

Output
-
******************************************************************************)
METHOD PROTECTED writeBuffer : ERetCode_t
VAR_INPUT
END_VAR
VAR
	u32Len : UDINT;
END_VAR

	writeBuffer := eRetCode_t.eRetBusy;
	
	IF LEN(strBuffer) <= 0 THEN
		RETURN;
	END_IF
	
	u32Len := TO_UDINT(LEN(strBuffer)); 
	
	writeBuffer := writeData(i_pData := ADR(strBuffer), u32Size := u32Len);
END_METHOD

(******************************************************************************
Baustein: FB_TestReportBase.writeData
Spezifikation: doc/Spezifikation.pdf, Kap. x.y.z
-------------------------------------------------------------------------------
erstellt:
von:
Geändert:
von:
-------------------------------------------------------------------------------
Beschreibung


-------------------------------------------------------------------------------
Input
	i_pData : POINTER TO BYTE;
	u32Size : UDINT;
	
Output
-
******************************************************************************)
METHOD PROTECTED writeData : ERetCode_t
VAR_INPUT
	i_pData : POINTER TO BYTE;
	u32Size : UDINT;
END_VAR

	writeData := ERetCode_t.eRetFailed;
	
	IF u32Size = 0 OR i_pData = 0 THEN
		RETURN;
	END_IF
	
	fbWrite.pWriteBuff 	:= i_pData; 
	fbWrite.cbWriteLen 	:= u32Size; 
	fbWrite.hFile 		:= fbOpen.hFile; 
	fbWrite.bExecute 	:= TRUE;
			
	IF trgWrite.Q = TRUE THEN
		writeData := ERetCode_t.eRetDone;
		fbWrite.bExecute 	:= FALSE;			
	ELSE	
		writeData := ERetCode_t.eRetBusy;
	END_IF;	

	IF fbWrite.bError = TRUE THEN
		writeData := eRetCode_t.eRetFailed;
	END_IF;
END_METHOD

END_FUNCTION_BLOCK

// ---- Test/FB_Test_Base.TcPOU
FUNCTION_BLOCK FB_Test_Base EXTENDS FB_UnitTestBase
VAR_INPUT
END_VAR
VAR_OUTPUT
END_VAR
VAR
END_VAR

(******************************************************************************
Baustein: FB_UnitTestBase.cleanup
Spezifikation: doc/Spezifikation.pdf, Kap. x.y.z
-------------------------------------------------------------------------------
erstellt:
von:
Geändert:
von:
-------------------------------------------------------------------------------
Beschreibung
Diese Methode...

-------------------------------------------------------------------------------
Input
-

Output
-
******************************************************************************)
METHOD PUBLIC cleanup : BOOL
VAR_INPUT
END_VAR

	cleanup := true;
END_METHOD

(******************************************************************************
Baustein: FB_Test_Base.execute
Spezifikation: doc/Spezifikation.pdf, Kap. x.y.z
-------------------------------------------------------------------------------
erstellt:
von:
Geändert:
von:
-------------------------------------------------------------------------------
Beschreibung
Diese Methode...

-------------------------------------------------------------------------------
Input
-

Output
-
******************************************************************************)
METHOD PUBLIC execute : BOOL
VAR_INPUT
END_VAR
VAR
	bValue1  : BOOL;
	bValue2  : BOOL;
	s32Value1 : DINT;
	s32Value2 : DINT;
	r32Value1 : REAL;
	r32Value2 : REAL;
END_VAR

	bValue1 := TRUE;
	bValue2 := TRUE;
	assertEQUAL(bValue1, bValue2);

	s32Value1 := 1593;
	s32Value2 := 1593;
	assertEQUAL(s32Value1, s32Value2);

	r32Value1 := 5345.53245;
	r32Value2 := 5345.53245;
	assertEQUAL(r32Value1, r32Value2);

	execute := TRUE;
END_METHOD

(******************************************************************************
Baustein: FB_UnitTestBase.prepare
Spezifikation: doc/Spezifikation.pdf, Kap. x.y.z
-------------------------------------------------------------------------------
erstellt:
von:
Geändert:
von:
-------------------------------------------------------------------------------
Beschreibung
Diese Methode...

-------------------------------------------------------------------------------
Input
-

Output
-
******************************************************************************)
METHOD PUBLIC prepare : BOOL
VAR_INPUT
END_VAR

	prepare := true;
END_METHOD

END_FUNCTION_BLOCK

// ---- Test/FB_Test_Base_Delay.TcPOU
{attribute 'hide'}
FUNCTION_BLOCK FB_Test_Base_Delay EXTENDS FB_TestBase
VAR_INPUT
END_VAR
VAR_OUTPUT
END_VAR
VAR
	fbDelay : TON;
END_VAR

(******************************************************************************
Baustein: FB_Test_Base_Delay.cleanup
Spezifikation: doc/Spezifikation.pdf, Kap. x.y.z
-------------------------------------------------------------------------------
erstellt:
von:
Geändert:
von:
-------------------------------------------------------------------------------
Beschreibung
Diese Methode...

-------------------------------------------------------------------------------
Input
-

Output
-
******************************************************************************)
METHOD PUBLIC cleanup : ERetCode_t
VAR_INPUT
END_VAR

	cleanup := ERetCode_t.eRetDone;
	
	fbDelay(IN := false);
END_METHOD

(******************************************************************************
Baustein: FB_Test_Base_Delay.execute
Spezifikation: doc/Spezifikation.pdf, Kap. x.y.z
-------------------------------------------------------------------------------
erstellt:
von:
Geändert:
von:
-------------------------------------------------------------------------------
Beschreibung
Diese Methode...

-------------------------------------------------------------------------------
Input
-

Output
-
******************************************************************************)
METHOD PUBLIC execute : ERetCode_t
VAR_INPUT
END_VAR
VAR
	bValue1  : BOOL;
	bValue2  : BOOL;
	s32Value1 : DINT;
	s32Value2 : DINT;
	r32Value1 : REAL;
	r32Value2 : REAL;
END_VAR

	fbDelay(PT := t#250ms);
	execute 	  := ERetCode_t.eRetBusy;

	bValue1 := TRUE;
	bValue2 := TRUE;
	assert.EQUAL(bValue1, bValue2);

	s32Value1 := 1593;
	s32Value2 := 1593;
	assert.EQUAL(s32Value1, s32Value2);

	r32Value1 := 5345.53245;
	r32Value2 := 5345.53245;
	assert.EQUAL(r32Value1, r32Value2);

	if fbDelay.Q then
		execute := ERetCode_t.eRetDone;
	end_if;
END_METHOD

(******************************************************************************
Baustein: FB_Test_Base_Delay.prepare
Spezifikation: doc/Spezifikation.pdf, Kap. x.y.z
-------------------------------------------------------------------------------
erstellt:
von:
Geändert:
von:
-------------------------------------------------------------------------------
Beschreibung
Diese Methode...

-------------------------------------------------------------------------------
Input
-

Output
-
******************************************************************************)
METHOD PUBLIC prepare : ERetCode_t
VAR_INPUT
END_VAR

	prepare := ERetCode_t.eRetDone;
	
	fbDelay.IN := true;
END_METHOD

END_FUNCTION_BLOCK
